PROGRAM MAIN
VAR
	fb_SecPulse						: DFB_Second_Pulse;
	fbDel							: FB_Delay;
	fbDebugStationProcess			: FB_DebugStationProcess;
	fbDBStnUpdateStatus				: FB_DBStnUpdateStatus;
	fbTCMLevelEPTUpdate				: FB_TCMLevelEPTUpdate;
	fbGUI_TEST						: ARRAY [1..NO_OF_LEVEL] OF FB_GUI_TEST;
	fbGUI_TEST_SLTC					: ARRAY [1..NO_OF_LEVEL] OF FB_GUI_TEST_SLTC;
	fbUpdateStatus					: ARRAY [1..NO_OF_LEVEL] OF FB_UpdateStatus;
	fbTCShuttlePOC_Process			: ARRAY [1..NO_OF_LEVEL] OF FB_TCShuttlePOC_Process;
	fbTCMultiLevel_Process			: ARRAY [1..NO_OF_LEVEL] OF FB_TCMultiLevel_Process;
	fbTCLevel_Process				: ARRAY [1..NO_OF_LEVEL] OF FB_TCLevel_Process;
	
	bFbDelIn						: BOOL;	//Int for 20 Sec
	bFBDelOut						: BOOL;	//Int for 20 Sec
    bDebugging						: BOOL;	
	bDebug							: BOOL;
	bTemp							: BOOL;
	bForceFalse						: BOOL	:= FALSE;
	bErrorTemp						: BOOL;
	isDbStnTIIAlarm					: BOOL;
	DBColumnAlarmLED				: BOOL;
	
	isTIIAlarms						: ARRAY[1..NO_OF_LEVEL] OF BOOL;
	_TIIAlarmLED					: ARRAY[1..NO_OF_LEVEL] OF BOOL;
	_TIIAlarmEPT					: ARRAY[1..NO_OF_LEVEL] OF BOOL;
	bAlarmBlock						: ARRAY[1..NO_OF_LEVEL] OF BOOL;
	
	
	_iSubModToRset					: INT;	//Get From TA Command
	_iAlmIDToRset					: INT;	//Get From TA Command
	
	noOfLevel						: UINT	:= 1;
	iLevel							: UINT;
	
	iUnBlock						: ARRAY[1..NO_OF_LEVEL] OF DINT;
	
	DbStnDIFU						: R_TRIG;
	DIFU							: ARRAY[1..NO_OF_LEVEL] OF R_TRIG;
	UnblockTIIDIFU					: ARRAY[1..NO_OF_LEVEL] OF R_TRIG;
	
	DbStnDIFD						: F_TRIG;
	DIFD							: ARRAY[1..NO_OF_LEVEL] OF F_TRIG;
	UnblockTIIDIFD					: ARRAY[1..NO_OF_LEVEL] OF F_TRIG;
	
	stTCMainVIO						: ST_TCColumn_VIO;
	stTCShuttlePOC_VIO				: ST_TCShuttlePOC_VIO;
	stTCMLevelVIO					: ST_TCMultiLevel_VIO;
	stDbStnVIO						: ST_DebugStation_VIO;
	
	//fbCommandEventMonitor : FB_CommandEventMonitor;
	
	
	
	
	
	
	
	fbTCMain						: INT;
	
	TestDIFU						: R_TRIG;
	
	iTestIntIndex					: INT;
	varBool							: BOOL;


	
	stDbColVIO						: ST_DebugColumnVIO;
	
	fb_Testing						: Testing;
END_VAR

///////////////////////////////////////////////////////////////////////////////////////////////////////////////////////////////////////////////////////////////////////////////////////////////////////////////////////////
//////////////////////////////////// Diagnostic mode configuration mapping //////////////////////////////////////////////////////////
///////////////////////////////////////////////////////////////////////////////////////////////////////////////////////////////////////////////////////////////////////////////////////////////////////////////////////////
stDbStnVIO 																	:= stDebugStation.fbDBStnSeq.P_stVIO;
stDbStnVIO.bDiagnosticMode													:= bDiagnosticMode;
stDebugStation.fbDBStnSeq.P_stVIO											:= stDbStnVIO;

stDbColVIO 																	:= fbDebugColumn.P_stVIO;
stDbColVIO.bDiagnosticMode 													:= bDiagnosticMode;
fbDebugColumn.P_stVIO														:= stDbColVIO;
	
///////////////////////////////////////////////////////////////////////////////////////////////////////////////////////////////////////////////////////////////////////////////////////////////////////////////////////////
///////////////////////////////	Always call /////////////////////////////////////////////////////////////////////////////////////////////
///////////////////////////////////////////////////////////////////////////////////////////////////////////////////////////////////////////////////////////////////////////////////////////////////////////////////////////
fb_SecPulse(TON1_TIME:= T#1S, QSec_P=> Sec_P);
PreInitialise();
ASSIGN_COLUMN();	// Get local Net ID to verify column ID

IF (NOT IsNetIDReadOK) AND bProductionMode THEN
	; //Reply Column Assignment Failed Event To TA
ELSE
/////////////////////////////////////////////////////////////////////////////////////////////////////////////////////////////////////////////////////////////////////////////////////////////////////////////////////////////////
/////////////////////////////// Debug Station /////////////////////////////////////////////////////////////////////////////////////////////
/////////////////////////////////////////////////////////////////////////////////////////////////////////////////////////////////////////////////////////////////////////////////////////////////////////////////////////////////
	IF bDebugStation THEN
		fbDBStnUpdateStatus(
			DBColumnAlarmLED			:= DBColumnAlarmLED
		);
		fbDebugColumn(
			DBColumnAlarmLED			=> DBColumnAlarmLED
		);	//Facility
		fbDebugStationProcess();	//Debug Station
		
		fbDbStnTIIAlarm(
			vIO																:= stDbStnVIO, 
			NoOfTIIAlm														:= NO_OF_TII_SENSOR, 
			iLevel															:= 1, (*stAlmMod:= ALMTC,*) 
			isTIIError														=> isDbStnTIIAlarm);
		
		DbStnDIFU(CLK:=isDbStnTIIAlarm);
		IF DbStnDIFU.Q THEN 
			stDbStnVIO														:= stGblDbStnVIO;
			stDbStnVIO.isTIIError											:= TRUE;	// To Ckeck the Bit In Process!
			stDebugStation.fbDBStnSeq.P_stVIO								:= stDbStnVIO;
		END_IF
		
		DbStnDIFD(CLK:=isDbStnTIIAlarm);
		IF DbStnDIFD.Q THEN 
			stDbStnVIO														:= stGblDbStnVIO;
			stDbStnVIO.isTIIError											:= FALSE;
			stDebugStation.fbDBStnSeq.P_stVIO								:= stDbStnVIO;
		END_IF
/////////////////////////////////////////////////////////////////////////////////////////////////////////////////////////////////////////////////////////////////////////////////////////////////////////////////////////////////
/////////////////////////////// TC & Full Cell Stack /////////////////////////////////////////////////////////////////////////////////////////////
/////////////////////////////////////////////////////////////////////////////////////////////////////////////////////////////////////////////////////////////////////////////////////////////////////////////////////////////////
	ELSE 
		fbSLTCExtra(); // Extra SLTC IO check;
		noOfLevel															:= SEL(bDebugCart, NO_OF_LEVEL, NO_OF_DC_CELL_LEVEL);
	
		FOR iLevel := 1 TO noOfLevel DO
			fbTCColumn(
				iLevel														:= iLevel);
				
			fbUpdateStatus[iLevel](
				iLevel														:= iLevel);
			
			fbTCColumn.M_UpdateSysAlarmFlag(
				iLevel														:= iLevel);
				
			fbTCMultiLevel_Process[iLevel](
				iLevel														:= iLevel);
				
			arrTCMultiLevelVIO[iLevel]										:= arrTCMultiLevel[iLevel].fbTCMultiLevelSeq.P_stTCMultiLevelVIO;
			
			fbTCMLevelEPTUpdate(
				iLevel														:= iLevel); //Update EPT State;
				
			stTCMLevelVIO													:= arrTCMultiLevelVIO[iLevel];
			bFbDelIn														:= stTCMLevelVIO.ipTesterPresent AND stTCMLevelVIO.ipTesterLatchesClosed;
			
			fbDel(
				msec														:= 20000,
				in															:= bFbDelIn,
				out															:= bFBDelOut);
			
			stTCMLevelVIO.bTstDelInt										:= bFBDelOut;
			arrTCMultiLevel[iLevel].fbTCMultiLevelSeq.P_stTCMultiLevelVIO	:= stTCMLevelVIO;
			
			// Update TIIAlarms
			arrTIIAlarm[iLevel](
				vIO																			:= arrTCMultiLevelVIO[iLevel],
				NoOfTIIAlm																	:= NO_OF_TII_SENSOR,
				iLevel																		:= iLevel, (*stAlmMod:= ALMTC,*)
				isTIIError																	=> isTIIAlarms[iLevel],
				iUnBlock																	=> iUnBlock[iLevel], 
				bAlarmBlock																	=> bAlarmBlock[iLevel],
				TIIAlarmLED																	=> _TIIAlarmLED[iLevel],
				TIIAlarmEPT																	=> _TIIAlarmEPT[iLevel]
			);
				
			stTCMLevelVIO 																:= arrTCMultiLevel[iLevel].fbTCMultiLevelSeq.P_stTCMultiLevelVIO;	
		
			IF stTCMLevelVIO.iUnBlock <> iUnBlock[iLevel] THEN
				stTCMLevelVIO.iUnBlock													:= iUnBlock[iLevel];
				arrTCMultiLevel[iLevel].fbTCMultiLevelSeq.P_stTCMultiLevelVIO			:= stTCMLevelVIO;
			END_IF
			
			IF stTCMLevelVIO.bAlarmBlock <> bAlarmBlock[iLevel] THEN
				stTCMLevelVIO.bAlarmBlock												:= bAlarmBlock[iLevel];
				arrTCMultiLevel[iLevel].fbTCMultiLevelSeq.P_stTCMultiLevelVIO			:= stTCMLevelVIO;
			END_IF
			
			IF stTCMLevelVIO.TIIAlarmEPT <> _TIIAlarmEPT[iLevel] THEN
				stTCMLevelVIO.TIIAlarmEPT												:= _TIIAlarmEPT[iLevel];
				arrTCMultiLevel[iLevel].fbTCMultiLevelSeq.P_stTCMultiLevelVIO			:= stTCMLevelVIO;
			END_IF
			
			IF stTCMLevelVIO.TIIAlarmLED <> _TIIAlarmLED[iLevel] THEN
				stTCMLevelVIO.TIIAlarmLED												:= _TIIAlarmLED[iLevel];
				arrTCMultiLevel[iLevel].fbTCMultiLevelSeq.P_stTCMultiLevelVIO			:= stTCMLevelVIO;
			END_IF
						
			DIFU[iLevel](CLK := isTIIAlarms[iLevel]);
			
			IF DIFU[iLevel].Q THEN 
				stTCMLevelVIO															:= arrTCMultiLevelVIO[iLevel];
				stTCMLevelVIO.isTIIError												:= TRUE; // To Ckeck the Bit In Process!
				//arrTCMultiLevelVIO[iLevel]:=stTCMLevelVIO;
				arrTCMultiLevel[iLevel].fbTCMultiLevelSeq.P_stTCMultiLevelVIO			:= stTCMLevelVIO;
			END_IF
			DIFD[iLevel](CLK := isTIIAlarms[iLevel]);
			IF DIFD[iLevel].Q THEN 
				stTCMLevelVIO															:= arrTCMultiLevelVIO[iLevel];
				stTCMLevelVIO.isTIIError												:= FALSE;
				//arrTCMultiLevelVIO[iLevel]:=stTCMLevelVIO;
				arrTCMultiLevel[iLevel].fbTCMultiLevelSeq.P_stTCMultiLevelVIO			:= stTCMLevelVIO;
			END_IF
			
			//Convert Int to Boolean 
			//EAP FROM TC => TBOT
			stTCMLevelVIO := arrTCMultiLevel[iLevel].fbTCMultiLevelSeq.P_stTCMultiLevelVIO;
			CASE iLevel OF
				1 :	
					stEAP.stTBOT_TC_EAP[iTCColumnID].iTCDrawerCylExtendRS_EAP.0		:= stTCMLevelVIO.ipTCDrawerCylExtendRS;
				2 :	
					stEAP.stTBOT_TC_EAP[iTCColumnID].iTCDrawerCylExtendRS_EAP.1		:= stTCMLevelVIO.ipTCDrawerCylExtendRS;
				3 :	
					stEAP.stTBOT_TC_EAP[iTCColumnID].iTCDrawerCylExtendRS_EAP.2		:= stTCMLevelVIO.ipTCDrawerCylExtendRS;
				4 :	
					stEAP.stTBOT_TC_EAP[iTCColumnID].iTCDrawerCylExtendRS_EAP.3		:= stTCMLevelVIO.ipTCDrawerCylExtendRS;
				5 :	
					stEAP.stTBOT_TC_EAP[iTCColumnID].iTCDrawerCylExtendRS_EAP.4		:= stTCMLevelVIO.ipTCDrawerCylExtendRS;
				6 :	
					stEAP.stTBOT_TC_EAP[iTCColumnID].iTCDrawerCylExtendRS_EAP.5		:= stTCMLevelVIO.ipTCDrawerCylExtendRS;
			END_CASE
				
			CASE iLevel OF
				1 :	
					stEAP.stTBOT_TC_EAP[iTCColumnID].iTCDrawerCylRetractRS_EAP.0	:= stTCMLevelVIO.ipTCDrawerCylRetractRS;
				2 :	
					stEAP.stTBOT_TC_EAP[iTCColumnID].iTCDrawerCylRetractRS_EAP.1	:= stTCMLevelVIO.ipTCDrawerCylRetractRS;
				3 :	
					stEAP.stTBOT_TC_EAP[iTCColumnID].iTCDrawerCylRetractRS_EAP.2	:= stTCMLevelVIO.ipTCDrawerCylRetractRS;
				4 :	
					stEAP.stTBOT_TC_EAP[iTCColumnID].iTCDrawerCylRetractRS_EAP.3	:= stTCMLevelVIO.ipTCDrawerCylRetractRS;
				5 :	
					stEAP.stTBOT_TC_EAP[iTCColumnID].iTCDrawerCylRetractRS_EAP.4	:= stTCMLevelVIO.ipTCDrawerCylRetractRS;
				6 :	
					stEAP.stTBOT_TC_EAP[iTCColumnID].iTCDrawerCylRetractRS_EAP.5	:= stTCMLevelVIO.ipTCDrawerCylRetractRS;
			END_CASE	
				
				//EAP FROM TBOT => TC
			CASE iLevel OF		
				1 :	
					varBool															:= stEAP.stTBOT_TC_EAP[iTCColumnID].iTCDwrSafeToMoveEAP.0;
				2 :	
					varBool															:= stEAP.stTBOT_TC_EAP[iTCColumnID].iTCDwrSafeToMoveEAP.1;
				3 :	
					varBool															:= stEAP.stTBOT_TC_EAP[iTCColumnID].iTCDwrSafeToMoveEAP.2;
				4 :	
					varBool															:= stEAP.stTBOT_TC_EAP[iTCColumnID].iTCDwrSafeToMoveEAP.3;
				5 :	
					varBool															:= stEAP.stTBOT_TC_EAP[iTCColumnID].iTCDwrSafeToMoveEAP.4;
				6 :	
					varBool															:= stEAP.stTBOT_TC_EAP[iTCColumnID].iTCDwrSafeToMoveEAP.5;
			END_CASE
	        
			stEAP.arrTBOT_TC_SubLevelEAP[iTCColumnID,iLevel].bTCDwrSafeToMoveEAP	:= varBool;
			
			//<Convert Int to Bool>
			//TBOT => TC
			//arrTCMultiLevel[i].stGblParam.iTCDwrSafeToMoveEAP := stEAP.arrTBOT_TC_SubLevelEAP[iTCColumnID,iLevel].iTCDwrSafeToMoveEAP;	//arrTCDwrSafeToMoveEAP[iLevel];
			arrTCMultiLevel[iLevel].stGblParam.bTCDwrSafeToMoveEAP 						:= stEAP.arrTBOT_TC_SubLevelEAP[iTCColumnID,iLevel].bTCDwrSafeToMoveEAP;	//stEAP.stTBOT_TC_EAP[iTCColumnID].iTCDwrSafeToMoveEAP;//.arrTCDwrSafeToMoveEAP[iLevel];	
			arrTCMultiLevel[iLevel].stGblParam.bTBotAntiCollisionTriggered				:= stEAP.stTBOT_TC_EAP[iTCColumnID].bAntiCollisionTriggered;	//stEAP_TC_TBOT.bAntiCollisionTriggered;
			arrTCMultiLevel[iLevel].stGblParam.bTCCellACPwrOff							:= stEAP.stTBOT_TC_EAP[iTCColumnID].bTCCellACPwrOff;	//stEAP_TC_TBOT.bAntiCollisionTriggered;
			arrTCMultiLevel[iLevel].fbTCMultiLevelSeq.P_stParam							:= arrTCMultiLevel[iLevel].stGblParam;	//set value
		END_FOR
	END_IF	
END_IF	

CmdAndEventProcess();
Logging();
TestManually();

////////////////////////////////////////////////////////////////////////////////////////////////////////////////////////////////////////////////////////////////////////////////////////////////////////////////////////////////////
/////////////////////////////////////// For Troubleshooting Purpose ///////////////////////////////////////
////////////////////////////////////////////////////////////////////////////////////////////////////////////////////////////////////////////////////////////////////////////////////////////////////////////////////////////////////
TestDIFU(clk := ALMTC.Level[1].AlarmID[4]);

IF TestDIFU.Q THEN 
	;//for troubleshooting
END_IF

// Jimmy Testing Purpose
fb_Testing();

END_PROGRAM

(* stored: Version 1.1.0.1, ProductVersion 3.1.4022.18
   POU MAIN: Id {aae7410b-55c4-4d1b-8483-7c04414fd9ab}, SpecialFunc None *)
